Universal Robots PolyScope program: demo_pick_and_place_with_subprograms.urp

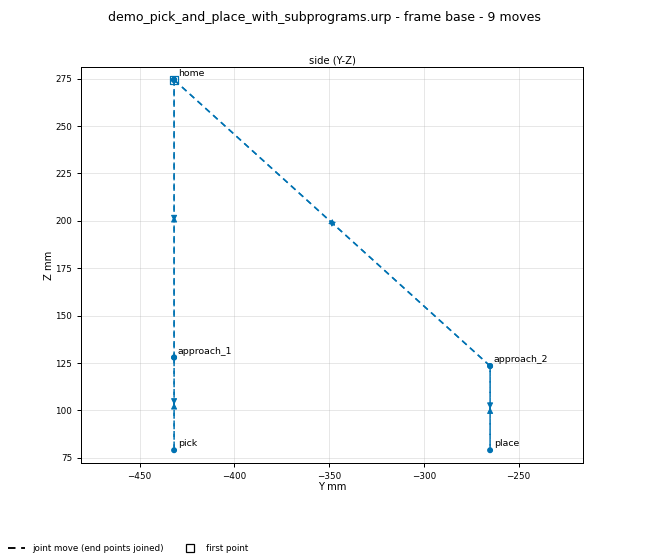
[picture p0: tool path of demo_pick_and_place_with_subprograms.urp in frame base, 9 of 9 moves have a stored position in this frame; points joined in program order, loops and branches not executed]
ProgramRoot setBeforeStartSequence=true; setInitialVariableValues=true; directory=/home/ur/ursim-1.8/programs/robotiq_3f_gripper_programs; kinematics=(a=[0, -0.425, -0.39225, 0, 0, 0], d=[0.08916, 0, 0, 0.10915, 0.09465, 0.0823], alpha=[1.5708, 0, 0, 1.5708, -1.5708, 0], deltaTheta=[0, 0, 0, 0, 0, 0], status=notInitialized); name=demo_pick_and_place_with_subprograms; robotEnvironmentFileName=rq_3FG
  InitVariables 
  BeforeStart description=COMMAND_SEQUENCE_BEFORE_PROGRAM_START; name=BeforeStart
    Script type=1; cachedFileContents=################################################################
      | ## Script file used to communicate with Robotiq's 3F Gripper 
      | ## Version: 2.0.0
      | ################################################################
      | 
      | # aliases for the gripper output names
      | # those values also represent offsets 
      | # in control registers
      | rACT = 1
      | rMOD = 2
      | rGTO = 8
      | rATR = 16
      | rPOS = 3
      | rFOR = 5
      | rSPE = 11
      | 
      | # aliases for the gripper input names
      | # those values also represent offsets 
      | # in control registers
      | gPRE = 1
      | gACT = 8
      | gMOD = 9
      | gMOD1 = 9
      | gMOD2 = 10
      | gFLT = 19
      | gFLT1 = 8
      | gFLT2 = 9
      | gFLT3 = 10
      | gFLT4 = 11
      | gGTO = 11
      | gIMC = 12
      | gIMC1 = 12
      | gIMC2 = 13
      | gSTA = 14
      | gSTA1 = 14
      | gSTA2 = 15
      | 
      | # send the activation request to the gripper.
      | def rq_activate():
      | 	rq_set_var(rACT,1)
      | 
      |     ACT = rq_get_var(gACT)
      |     while (ACT != 1):
      |         ACT = rq_get_var(gACT)
      |     end
      | end
      | 
      | # send the activation request to the gripper and
      | # wait for its completion.
      | def rq_activate_and_wait():
      | 	rq_activate()
      | 
      | 	while(not rq_is_gripper_activated()):
      | 		# wait for activation completed
      | 	end
      | end
      | 
      | # interrupts the gripper motion.
      | def rq_stop():
      | 	rq_set_var(rGTO,0)
      | 
      |     GTO = rq_get_var(gGTO)
      |     while (GTO != 0):
      |         GTO = rq_get_var(gGTO)
      |     end
      | end
      | 
      | # resets the activation and auto-release bits.
      | def rq_reset():
      | 	rq_set_var(rATR,0)
      | 	rq_set_var(rACT,0)
      | 
      |     ACT = rq_get_var(gACT)
      |     while (ACT != 0):
      |         ACT = rq_get_var(gACT)
      |     end
      | end
      | 
      | # send the auto-release request and wait 
      | # for its completion
      | def rq_auto_release_and_wait():
      | 	rq_set_var(rACT,1)
      | 	rq_set_var(rATR,1)
      | 
      |     ACT = rq_get_var(gACT)
      |     while (ACT != 1):
      |         ACT = rq_get_var(gACT)
      |     end
      | 
      | 	FLT = rq_get_var(gFLT)
      | 	while(FLT != 15):
      | 		FLT = rq_get_var(gFLT)
      | 	end
      | end
      | 
      | # set the force setpoint
      | def rq_set_force(force):
      | 	rq_set_var(rFOR,force)
      | end
      | 
      | # set the speed setpoint
      | def rq_set_speed(speed):
      | 	rq_set_var(rSPE,speed)
      | end
      | 
      | # send the open request to the gripper
      | def rq_open():
      | 	rq_move(0)
      | end
      | 
      | # send the close request to the gripper
      | def rq_close():
      | 	rq_move(255)
      | end
      | 
      | # send the open request to the gripper and wait
      | # for its completion
      | def rq_open_and_wait():
      | 	rq_move_and_wait(0)
      | end
      | 
      | # send the close request to the gripper and wait
      | # for its completion
      | def rq_close_and_wait():
      | 	rq_move_and_wait(255)
      | end
      | 
      | # send the move request to the position in argument
      | def rq_move(pos):
      | 	rq_set_var(rGTO,0)
      | 
      | 	GTO = rq_get_var(gGTO)
      | 	while (GTO != 0):
      | 		GTO = rq_get_var(gGTO)
      | 	end
      | 
      | 	rq_set_var(rPOS,pos)
      | 	
      | 	PRE = rq_get_var(gPRE)
      | 	while (PRE != pos):
      | 		PRE = rq_get_var(gPRE)
      | 	end
      | 
      | 	rq_set_var(rGTO,1)
      | 
      | 	while (GTO != 1):
      | 		GTO = rq_get_var(gGTO)
      | 	end
      | 		
      | end
      | 
      | # send the move request to the position in argument
      | # and wait for its completion
      | def rq_move_and_wait(pos):
      | 	rq_move(pos)
      | 
      | 	while (not rq_is_motion_complete()):
      | 		# wait for motion completed
      | 		sleep(0.01)
      | 		sync()
      | 	end
      | end
      | 
      | # send the request to change mode in argument
      | def rq_set_mode(value):
      | 	rq_set_var(rMOD, value)
      | 
      |     MOD = rq_get_var(gMOD)
      |     while (MOD != value):
      |         MOD = rq_get_var(gMOD)
      |     end
      | end
      | 
      | # send the request to change to the basic mode
      | def rq_set_basic_mode():
      | 	rq_set_mode(0)
      | end
      | 
      | # send the request to change to the pinch mode
      | def rq_set_pinch_mode():
      | 	rq_set_mode(1)
      | end
      | 
      | # send the request to change to the wide mode
      | def rq_set_wide_mode():
      | 	rq_set_mode(2)
      | end
      | 
      | # send the request to change to the scissor mode
      | def rq_set_scissor_mode():
      | 	rq_set_mode(3)
      | end
      | 
      | # returns True if the gripper has completed its motion
      | # returns False otherwise
      | def rq_is_motion_complete():
      | 	STA = rq_get_var(gSTA)
      | 
      | 	if (STA == 0):
      | 		return False
      | 	end
      | 
      | 	return True
      | 
      | end
      | 
      | # Returns True if the gripper is activated
      | def rq_is_gripper_activated():
      |     IMC = rq_get_var(gIMC)
      |     
      |     if (IMC == 3):
      |         return True
      |     end
      | 
      |     return False
      | end
      | 
      | # returns True if an object has been detected
      | def rq_is_object_detected():
      | 	STA = rq_get_var(gSTA)
      | 
      | 	if(STA == 1):
      | 		return True
      | 	elif(STA == 2):
      | 		return True
      | 	else:
      | 		return False
      | 	end
      | end
      | 
      | # prints in the log window the fault status
      | def rq_print_fault_code():
      | 	fault_status = rq_get_var(gFLT)
      | 
      | 	if(fault_status == 0):
      | 		textmsg("Gripper Fault : ", "No Fault (0x00)")
      | 	elif (fault_status == 5):
      | 		textmsg("Gripper Fault : ", "Priority Fault: Action delayed, activation (reactivation) must be completed prior to renewed action (0x05)")
      | 	elif (fault_status == 6):
      | 		textmsg("Gripper Fault : ", "Priority Fault: Action delayed, mode change must be completed prior to continuing action (0x06)")
      | 	elif (fault_status == 7):
      | 		textmsg("Gripper Fault : ", "Priority Fault: The activation bit must be set prior to action (0x07)")
      | 	elif (fault_status == 9):
      | 		textmsg("Gripper Fault : ", "Minor Fault: The communication chip is not ready (may be booting) (0x09)")
      | 	elif (fault_status == 10):
      | 		textmsg("Gripper Fault : ", "Minor Fault: Changing mode fault, interference detected on Scissor (for less than 20 sec) (0x0A)")
      | 	elif (fault_status == 11):
      | 		textmsg("Gripper Fault : ", "Minor Fault: Automatic release in progress (0x0B)")
      | 	elif (fault_status == 13):
      | 		textmsg("Gripper Fault : ", "Major Fault: Activation fault, verify that no interference or other error occurred (0x0D)")
      | 	elif (fault_status == 14):
      | 		textmsg("Gripper Fault : ", "Major Fault: Changing mode fault, interference detected on Scissor (for more than 20 sec) (0x0E)")
      | 	elif (fault_status == 15):
      | 		textmsg("Gripper Fault : ", "Major Fault: Automatic release completed. Reset and activation is required (0x0F)")
      | 	else:
      | 		textmsg("Gripper Fault : ", "Unkwown Fault")
      | 	end
      | end
      | 
      | # sets the gripper inputs
      | global current_force = 0
      | global current_speed = 0
      | def rq_set_var(name, value):
      | 	
      | 	if (name == rACT):
      |         MOD = rq_get_var(gMOD)
      |         GTO = rq_get_var(gGTO)
      |         modbus_set_output_register("gripper_O0", 256 * (rACT * value + rMOD * MOD + rGTO * GTO), False)
      | 	elif (name == rMOD):
      |         ACT = rq_get_var(gACT)
      |         GTO = rq_get_var(gGTO)
      |         modbus_set_output_register("gripper_O0", 256 * (rACT * ACT + rMOD * value + rGTO * GTO), False)
      | 	elif (name == rGTO):
      |         ACT = rq_get_var(gACT)
      |         MOD = rq_get_var(gMOD)
      |        	modbus_set_output_register("gripper_O0", 256 * (rACT * ACT + rMOD * MOD + rGTO * value), False)
      | 	elif (name == rATR):
      |         ACT = rq_get_var(gACT)
      |         MOD = rq_get_var(gMOD)
      |         GTO = rq_get_var(gGTO)
      |        	modbus_set_output_register("gripper_O0", 256 * (rACT * ACT + rMOD * MOD + rGTO * GTO + rATR * value), False)
      | 	elif (name == rFOR):
      |         current_force = value
      |         modbus_set_output_register("gripper_O2", (256 * current_speed + value), False)
      | 	elif (name == rSPE):
      |         current_speed = value
      |        	modbus_set_output_register("gripper_O2", (256 * value + current_force), False)
      | 	elif (name == rPOS):
      |         modbus_set_output_register("gripper_O1", value, False)
      |     else:
      |     end
      | 
      |     sync()
      | end
      | 
      | # reads the gripper outputs
      | def rq_get_var(name, nbr_bytes=0):
      |     if (name == gACT):
      |         reg = integer_to_binary_list(modbus_get_signal_status("gripper_I0", False))
      |         value = binary_list_to_integer([reg[gACT]])
      |     elif (name == gMOD):
      |         reg = integer_to_binary_list(modbus_get_signal_status("gripper_I0", False))
      |         value = binary_list_to_integer([reg[gMOD1], reg[gMOD2]])
      |     elif (name == gGTO):
      |         reg = integer_to_binary_list(modbus_get_signal_status("gripper_I0", False))
      |         value = binary_list_to_integer([reg[gGTO]])
      |     elif (name == gSTA):
      |         reg = integer_to_binary_list(modbus_get_signal_status("gripper_I0", False))
      |         value = binary_list_to_integer([reg[gSTA1], reg[gSTA2]])
      |     elif (name == gIMC):
      |         reg = integer_to_binary_list(modbus_get_signal_status("gripper_I0", False))
      |         value = binary_list_to_integer([reg[gIMC1], reg[gIMC2]])
      |     elif (name == gFLT):
      |         reg = integer_to_binary_list(modbus_get_signal_status("gripper_I1", False))
      |         value = binary_list_to_integer([reg[gFLT1], reg[gFLT2], reg[gFLT3], reg[gFLT4]])
      |     elif (name == gPRE):
      |         reg = modbus_get_signal_status("gripper_I1", False)
      |         value = reg % 256
      |     else:
      |    	    value = 0
      |     end
      |      
      |     sync()
      | 
      |     return value
      | end; scriptFile=/home/ur/ursim-1.8/programs/robotiq_3f_gripper_programs/rq_3FG_api.script
    Assignment assignmentValueSource=0; expr=0; operatorValueType=INTEGER; valueSource=EXPRESSION; variable=0
    Assignment assignmentValueSource=0; expr=255; operatorValueType=INTEGER; valueSource=EXPRESSION; variable=0
  MainProgram cartesianAcceleration=1.2; cartesianSpeed=0.25; jointAcceleration=1.3962634015954636; jointSpeed=1.0471975511965976; moveAsFastAsPossible=true; sharedProcessMoveBlendRadius=0.025; featureReference=(installationNameReference=Base); motionType=JOINT_SPACE; runOnlyOneCycle=true
    Comment commentString=This program moves the robot to an object.
    Comment commentString=It then picks it and moves it to another
    Comment commentString=location.
    CallSubProgram subProgramNodeToCall=rq_set_force(rq_force)
    CallSubProgram subProgramNodeToCall=rq_set_speed(rq_speed)
    CallSubProgram subProgramNodeToCall=rq_activate_and_wait()
    CallSubProgram subProgramNodeToCall=rq_open_and_wait()
    Move cartesianAcceleration=1.2; cartesianSpeed=0.25; jointAcceleration=1.3962634015954636; jointSpeed=1.0471975511965976; moveAsFastAsPossible=true; sharedProcessMoveBlendRadius=0.025; featureReference=(installationNameReference=Base); motionType=JOINT_SPACE
      Waypoint blendRadius=0.05; cartesianAcceleration=1.2; cartesianSpeed=0.25; jointAcceleration=1.3962634015954636; jointSpeed=1.0471975511965976; nextMotionTime=2.0; stoppoint=true; useSharedBlendParameter=true; useSharedParameters=true; position=TCP in base x=-120.113 y=-431.761 z=274.386 mm, rx=-0.0012 ry=3.1163 rz=0.0389 rad; joints [-91.713, -87.601, -115.63, -68.242, 91.392, -1.776] deg; positionType=FIXED_POSITION; waypointPoseInFeatureCoordinates=(pos=(x=-0.1201130103353891, y=-0.4317606580015477, z=0.2743855757605886), rot=(x=-0.00122135968159332, y=3.116276528481954, z=0.038891915636889256)); name=home
      Waypoint blendRadius=0.05; cartesianAcceleration=1.2; cartesianSpeed=0.25; jointAcceleration=1.3962634015954636; jointSpeed=1.0471975511965976; nextMotionTime=2.0; stoppoint=true; useSharedBlendParameter=true; useSharedParameters=true; position=TCP in base x=-120.113 y=-431.758 z=127.919 mm, rx=-0.0012 ry=3.1163 rz=0.0389 rad; joints [-91.713, -101.182, -127.255, -43.036, 91.392, -1.776] deg; positionType=FIXED_POSITION; waypointPoseInFeatureCoordinates=(pos=(x=-0.12011292329006278, y=-0.4317577480118261, z=0.12791870504696637), rot=(x=-0.0012213596815903148, y=3.1162765284819804, z=0.03889191563687878)); name=approach_1
    Move cartesianAcceleration=1.2; cartesianSpeed=0.25; jointAcceleration=1.3962634015954636; jointSpeed=1.0471975511965976; moveAsFastAsPossible=true; sharedProcessMoveBlendRadius=0.025; featureReference=(installationNameReference=Base); motionType=JOINT_SPACE
      Waypoint blendRadius=0.05; cartesianAcceleration=1.2; cartesianSpeed=0.25; jointAcceleration=1.3962634015954636; jointSpeed=1.0471975511965976; nextMotionTime=2.0; stoppoint=true; useSharedBlendParameter=true; useSharedParameters=true; position=TCP in base x=-120.113 y=-431.755 z=78.977 mm, rx=-0.0012 ry=3.1163 rz=0.0389 rad; joints [-91.713, -107.888, -129.378, -34.208, 91.392, -1.776] deg; positionType=FIXED_POSITION; waypointPoseInFeatureCoordinates=(pos=(x=-0.12011283734170543, y=-0.4317548746946599, z=0.07897675599398006), rot=(x=-0.0012213596815881583, y=3.1162765284819804, z=0.03889191563688198)); name=pick
      CallSubProgram subProgramNodeToCall=rq_close_and_wait()
      Waypoint blendRadius=0.05; cartesianAcceleration=1.2; cartesianSpeed=0.25; jointAcceleration=1.3962634015954636; jointSpeed=1.0471975511965976; nextMotionTime=2.0; stoppoint=true; useSharedBlendParameter=true; useSharedParameters=true; position=TCP in base x=-120.113 y=-431.758 z=127.919 mm, rx=-0.0012 ry=3.1163 rz=0.0389 rad; joints [-91.713, -101.182, -127.255, -43.036, 91.392, -1.776] deg; positionType=FIXED_POSITION; waypointPoseInFeatureCoordinates=(pos=(x=-0.12011292329006278, y=-0.4317577480118261, z=0.12791870504696637), rot=(x=-0.0012213596815903148, y=3.1162765284819804, z=0.03889191563687878)); name=approach_1
    Move cartesianAcceleration=1.2; cartesianSpeed=0.25; jointAcceleration=1.3962634015954636; jointSpeed=1.0471975511965976; moveAsFastAsPossible=true; sharedProcessMoveBlendRadius=0.025; featureReference=(installationNameReference=Base); motionType=JOINT_SPACE
      Waypoint blendRadius=0.05; cartesianAcceleration=1.2; cartesianSpeed=0.25; jointAcceleration=1.3962634015954636; jointSpeed=1.0471975511965976; nextMotionTime=2.0; stoppoint=true; useSharedBlendParameter=true; useSharedParameters=true; position=TCP in base x=-120.113 y=-431.761 z=274.386 mm, rx=-0.0012 ry=3.1163 rz=0.0389 rad; joints [-91.713, -87.601, -115.63, -68.242, 91.392, -1.776] deg; positionType=FIXED_POSITION; waypointPoseInFeatureCoordinates=(pos=(x=-0.1201130103353891, y=-0.4317606580015477, z=0.2743855757605886), rot=(x=-0.00122135968159332, y=3.116276528481954, z=0.038891915636889256)); name=home
    CallSubProgram subProgramNodeToCall=rq_is_object_detected()
    If expr=not rq_is_object_detected(); type=IF_NODE
      Halt 
      Comment commentString=No object detected. Manage the case.
    Move cartesianAcceleration=1.2; cartesianSpeed=0.25; jointAcceleration=1.3962634015954636; jointSpeed=1.0471975511965976; moveAsFastAsPossible=true; sharedProcessMoveBlendRadius=0.025; featureReference=(installationNameReference=Base); motionType=JOINT_SPACE
      Waypoint blendRadius=0.05; cartesianAcceleration=1.2; cartesianSpeed=0.25; jointAcceleration=1.3962634015954636; jointSpeed=1.0471975511965976; nextMotionTime=2.0; stoppoint=true; useSharedBlendParameter=true; useSharedParameters=true; position=TCP in base x=-120.112 y=-265.033 z=123.405 mm, rx=-0.0012 ry=3.1163 rz=0.0389 rad; joints [-92.765, -79.764, -149.961, -41.774, 91.365, -2.827] deg; positionType=FIXED_POSITION; waypointPoseInFeatureCoordinates=(pos=(x=-0.1201119361337282, y=-0.2650331483718448, z=0.12340515561814756), rot=(x=-0.0012213597208201592, y=3.1162765274388784, z=0.038891917212786065)); name=approach_2
    Move cartesianAcceleration=1.2; cartesianSpeed=0.25; jointAcceleration=1.3962634015954636; jointSpeed=1.0471975511965976; moveAsFastAsPossible=true; sharedProcessMoveBlendRadius=0.025; featureReference=(installationNameReference=Base); motionType=JOINT_SPACE
      Waypoint blendRadius=0.05; cartesianAcceleration=1.2; cartesianSpeed=0.25; jointAcceleration=1.3962634015954636; jointSpeed=1.0471975511965976; nextMotionTime=2.0; stoppoint=true; useSharedBlendParameter=true; useSharedParameters=true; position=TCP in base x=-120.112 y=-265.042 z=78.974 mm, rx=-0.0012 ry=3.1163 rz=0.0389 rad; joints [-92.765, -90.253, -153.057, -28.188, 91.365, -2.827] deg; positionType=FIXED_POSITION; waypointPoseInFeatureCoordinates=(pos=(x=-0.12011236076304545, y=-0.2650419420708216, z=0.07897377284993704), rot=(x=-0.001221359720818002, y=3.116276527438878, z=0.0388919172127869)); name=place
      CallSubProgram subProgramNodeToCall=rq_open_and_wait()
      Waypoint blendRadius=0.05; cartesianAcceleration=1.2; cartesianSpeed=0.25; jointAcceleration=1.3962634015954636; jointSpeed=1.0471975511965976; nextMotionTime=2.0; stoppoint=true; useSharedBlendParameter=true; useSharedParameters=true; position=TCP in base x=-120.112 y=-265.033 z=123.405 mm, rx=-0.0012 ry=3.1163 rz=0.0389 rad; joints [-92.765, -79.764, -149.961, -41.774, 91.365, -2.827] deg; positionType=FIXED_POSITION; waypointPoseInFeatureCoordinates=(pos=(x=-0.1201119361337282, y=-0.2650331483718448, z=0.12340515561814756), rot=(x=-0.0012213597208201592, y=3.1162765274388784, z=0.038891917212786065)); name=approach_2
    Move cartesianAcceleration=1.2; cartesianSpeed=0.25; jointAcceleration=1.3962634015954636; jointSpeed=1.0471975511965976; moveAsFastAsPossible=true; sharedProcessMoveBlendRadius=0.025; featureReference=(installationNameReference=Base); motionType=JOINT_SPACE
      Waypoint blendRadius=0.05; cartesianAcceleration=1.2; cartesianSpeed=0.25; jointAcceleration=1.3962634015954636; jointSpeed=1.0471975511965976; nextMotionTime=2.0; stoppoint=true; useSharedBlendParameter=true; useSharedParameters=true; position=TCP in base x=-120.113 y=-431.761 z=274.386 mm, rx=-0.0012 ry=3.1163 rz=0.0389 rad; joints [-91.713, -87.601, -115.63, -68.242, 91.392, -1.776] deg; positionType=FIXED_POSITION; waypointPoseInFeatureCoordinates=(pos=(x=-0.1201130103353891, y=-0.4317606580015477, z=0.2743855757605886), rot=(x=-0.00122135968159332, y=3.116276528481954, z=0.038891915636889256)); name=home
  subProgramToCall [hidden by the author, left out]
  subProgramToCall [hidden by the author, left out]
  subProgramToCall [hidden by the author, left out]
  subProgramToCall [hidden by the author, left out]
  subProgramToCall [hidden by the author, left out]
  subProgramToCall [hidden by the author, left out]
